TYPE UR_O2T :
STRUCT
	IO:UR_8_O2T_Robot_IO;
	General_Register1:UR_9_O2T_Registers1;
	General_Register2:UR_9_O2T_Registers1;
END_STRUCT
END_TYPE

(* stored: Version 1.1.0.1
   DUT UR_O2T: Id {7ab39171-01ca-4447-9b5e-c40aa927a3cb} *)
